{attribute 'strict'}
{attribute 'qualified_only'}
TYPE E_CaseErectorMachineState :
(
	eIdle					:= 0,
	eAborting				:= 10,
	eAborted				:= 20,
	eStopping				:= 30,
	eStopped				:= 40,
	eStarting				:= 50,
	eRunning				:= 60,
	eReseting				:= 70,
	eRestarting				:= 80,
	eError					:= 1000	
);
END_TYPE

(* stored: Version 1.1.0.1, ProductVersion 3.1.4022.12
   DUT E_CaseErectorMachineState: Id {9da88e2f-a6c8-4589-9ac0-bb0f0652dfba} *)
